FUNCTION_BLOCK F_FROM_BIG_ENDIAN (* Convert from Big Endian *)
  (* Standard: 61131-3; Description: Copyright (c) 2013 TU Wien ACIN, HR Agrartechnik GmbH. This program and the accompanying materials are made available under the terms of the Eclipse Public License 2.0 which is available at https://www.eclipse.org/legal/epl-2.0/ SPDX-License-Identifier: EPL-2.0 Some portions generated by Gemini CLI *)
  (* Version 1.0, 2026-01-31, Franz Höpfinger, HR Agrartechnik GmbH, conform to IEC 61131-3 specification for this Block *)
  PACKAGE iec61131::conversion;
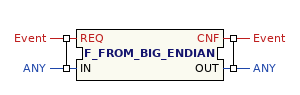
  EVENT_INPUT
    REQ WITH IN; (* Normal Execution Request *)
  END_EVENT
  EVENT_OUTPUT
    CNF WITH OUT; (* Execution Confirmation *)
  END_EVENT
  VAR_INPUT
    IN : ANY;
  END_VAR
  VAR_OUTPUT
    OUT : ANY;
  END_VAR
  EC_STATES
    REQ : REQ -> CNF;
  END_STATES
  ALGORITHM REQ IN ST:
OUT := FROM_BIG_ENDIAN(IN);
  END_ALGORITHM
END_FUNCTION_BLOCK
